// TIA Portal V20 export
TYPE "UDT_FIXTURE_IF"
   STRUCT
      Valves : Array[1..10] of "UDT_VALVE";
      PP : Array[1..35] of "PP_INTERFACE_UDT";
      Process_Complete : Array[1..16] of Bool;
      Work_Pos : Bool;
      Home_Pos : Bool;
      AtKnownPos : Bool;
   END_STRUCT;
END_TYPE
